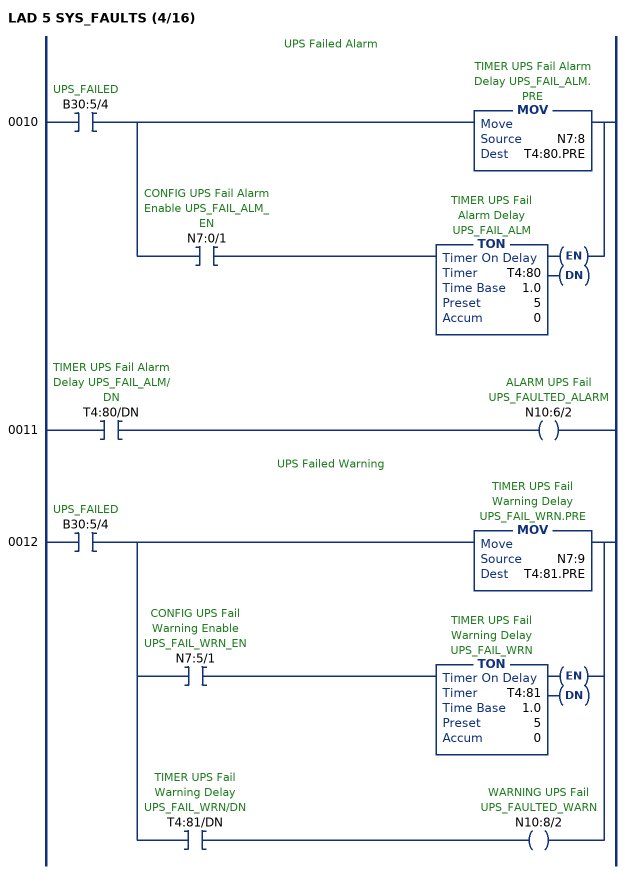
% Rung: 10 %
% UPS Failed Alarm %
SOR XIC B30:5/4 BST MOV N7:8 T4:80.PRE NXB XIC N7:0/1 TON T4:80 1.0 5 0 BND EOR
%   B30:5/4  UPS_FAILED %
%   N7:8  UPS_FAIL_ALM_DLY  "CONFIG UPS Fail Alarm Delay" %
%   T4:80  UPS_FAIL_ALM  "TIMER UPS Fail Alarm Delay" %
%   N7:0/1  UPS_FAIL_ALM_EN  "CONFIG UPS Fail Alarm Enable" %
% Rung: 11 %
SOR XIC T4:80/DN OTE N10:6/2 EOR
%   T4:80  UPS_FAIL_ALM  "TIMER UPS Fail Alarm Delay" %
%   N10:6/2  UPS_FAULTED_ALARM  "ALARM UPS Fail" %
% Rung: 12 %
% UPS Failed Warning %
SOR XIC B30:5/4 BST MOV N7:9 T4:81.PRE NXB XIC N7:5/1 TON T4:81 1.0 5 0 NXB XIC T4:81/DN OTE N10:8/2 BND EOR
%   B30:5/4  UPS_FAILED %
%   N7:9  UPS_FAIL_WRN_DLY  "CONFIG UPS Fail Warning Delay" %
%   T4:81  UPS_FAIL_WRN  "TIMER UPS Fail Warning Delay" %
%   N7:5/1  UPS_FAIL_WRN_EN  "CONFIG UPS Fail Warning Enable" %
%   N10:8/2  UPS_FAULTED_WARN  "WARNING UPS Fail" %

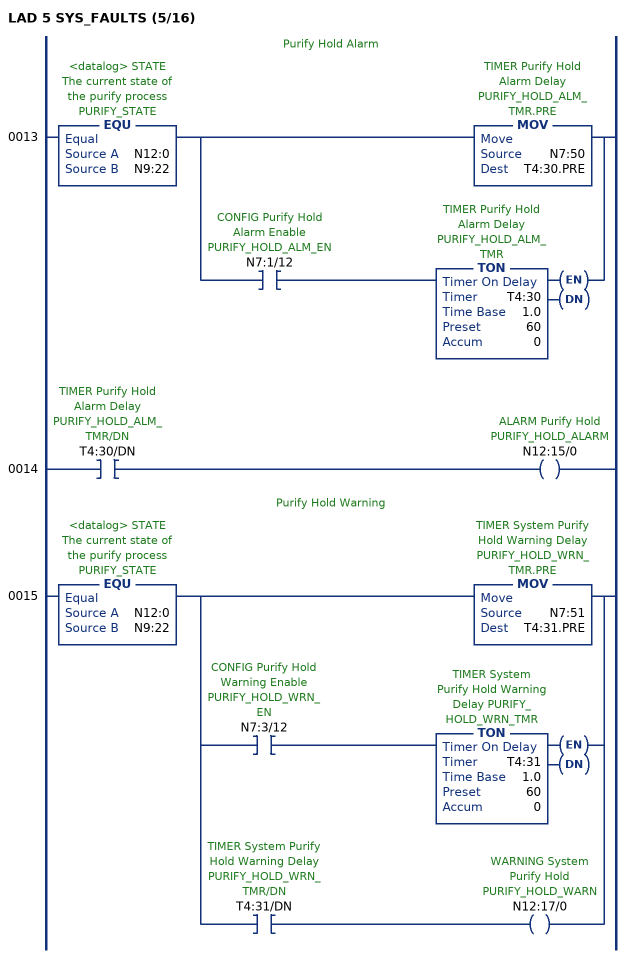
% Rung: 13 %
% Purify Hold Alarm %
SOR EQU N12:0 N9:22 BST MOV N7:50 T4:30.PRE NXB XIC N7:1/12 TON T4:30 1.0 60 0 BND EOR
%   N12:0  PURIFY_STATE  "<datalog> STATE The current state of the purify process" %
%   N9:22  PURIFY_HOLD  "STATE Purify Hold" %
%   N7:50  PURIFY_HOLD_ALM_DLY  "CONFIG Purify Hold Alarm Delay" %
%   T4:30  PURIFY_HOLD_ALM_TMR  "TIMER Purify Hold Alarm Delay" %
%   N7:1/12  PURIFY_HOLD_ALM_EN  "CONFIG Purify Hold Alarm Enable" %
% Rung: 14 %
SOR XIC T4:30/DN OTE N12:15/0 EOR
%   T4:30  PURIFY_HOLD_ALM_TMR  "TIMER Purify Hold Alarm Delay" %
%   N12:15/0  PURIFY_HOLD_ALARM  "ALARM Purify Hold" %
% Rung: 15 %
% Purify Hold Warning %
SOR EQU N12:0 N9:22 BST MOV N7:51 T4:31.PRE NXB XIC N7:3/12 TON T4:31 1.0 60 0 NXB XIC T4:31/DN OTE N12:17/0 BND EOR
%   N12:0  PURIFY_STATE  "<datalog> STATE The current state of the purify process" %
%   N9:22  PURIFY_HOLD  "STATE Purify Hold" %
%   N7:51  PURIFY_HOLD_WRN_DLY  "CONFIG Purify Hold Warning Delay" %
%   T4:31  PURIFY_HOLD_WRN_TMR  "TIMER System Purify Hold Warning Delay" %
%   N7:3/12  PURIFY_HOLD_WRN_EN  "CONFIG Purify Hold Warning Enable" %
%   N12:17/0  PURIFY_HOLD_WARN  "WARNING System Purify Hold" %

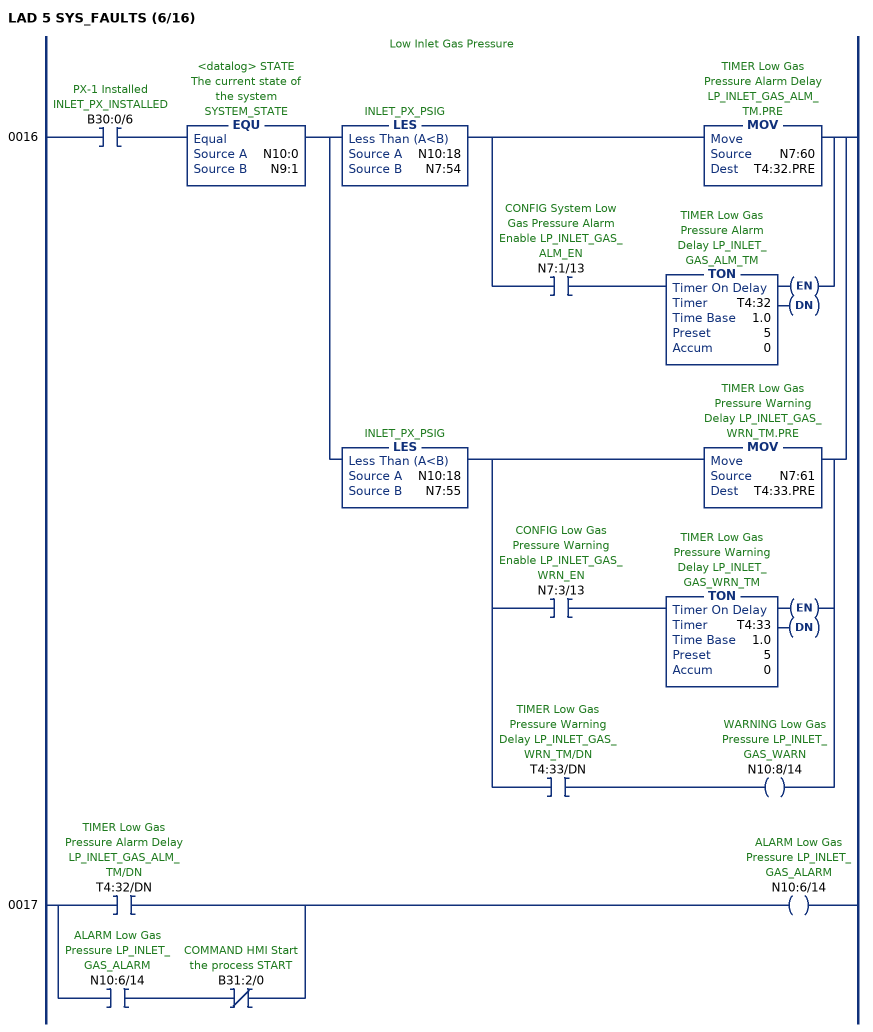
% Rung: 16 %
% Low Inlet Gas Pressure %
SOR XIC B30:0/6 EQU N10:0 N9:1 BST LES N10:18 N7:54 BST MOV N7:60 T4:32.PRE NXB XIC N7:1/13 TON T4:32 1.0 5 0 BND NXB LES N10:18 N7:55 BST MOV N7:61 T4:33.PRE NXB XIC N7:3/13 TON T4:33 1.0 5 0 NXB XIC T4:33/DN OTE N10:8/14 BND BND EOR
%   B30:0/6  INLET_PX_INSTALLED  "PX-1 Installed" %
%   N10:0  SYSTEM_STATE  "<datalog> STATE The current state of the system" %
%   N9:1  SYSTEM_PROCESS  "STATE System Process" %
%   N10:18  INLET_PX_PSIG %
%   N7:54  LP_INLET_GAS_ALM_SP  "CONFIG Gas Pressure Low Alarm Setpoint" %
%   N7:60  LP_INLET_GAS_ALM_DLY  "CONFIG Gas Pressure Low Alarm Delay" %
%   T4:32  LP_INLET_GAS_ALM_TM  "TIMER Low Gas Pressure Alarm Delay" %
%   N7:1/13  LP_INLET_GAS_ALM_EN  "CONFIG System Low Gas Pressure Alarm Enable" %
%   N7:55  LP_INLET_GAS_WRN_SP  "CONFIG Gas Pressure Low Warning Setpoint" %
%   N7:61  LP_INLET_GAS_WRN_DLY  "CONFIG Gas Pressure Low Warning Delay" %
%   T4:33  LP_INLET_GAS_WRN_TM  "TIMER Low Gas Pressure Warning Delay" %
%   N7:3/13  LP_INLET_GAS_WRN_EN  "CONFIG Low Gas Pressure Warning Enable" %
%   N10:8/14  LP_INLET_GAS_WARN  "WARNING Low Gas Pressure" %
% Rung: 17 %
SOR BST XIC T4:32/DN NXB XIC N10:6/14 XIO B31:2/0 BND OTE N10:6/14 EOR
%   T4:32  LP_INLET_GAS_ALM_TM  "TIMER Low Gas Pressure Alarm Delay" %
%   N10:6/14  LP_INLET_GAS_ALARM  "ALARM Low Gas Pressure" %
%   B31:2/0  START  "COMMAND HMI Start the process" %

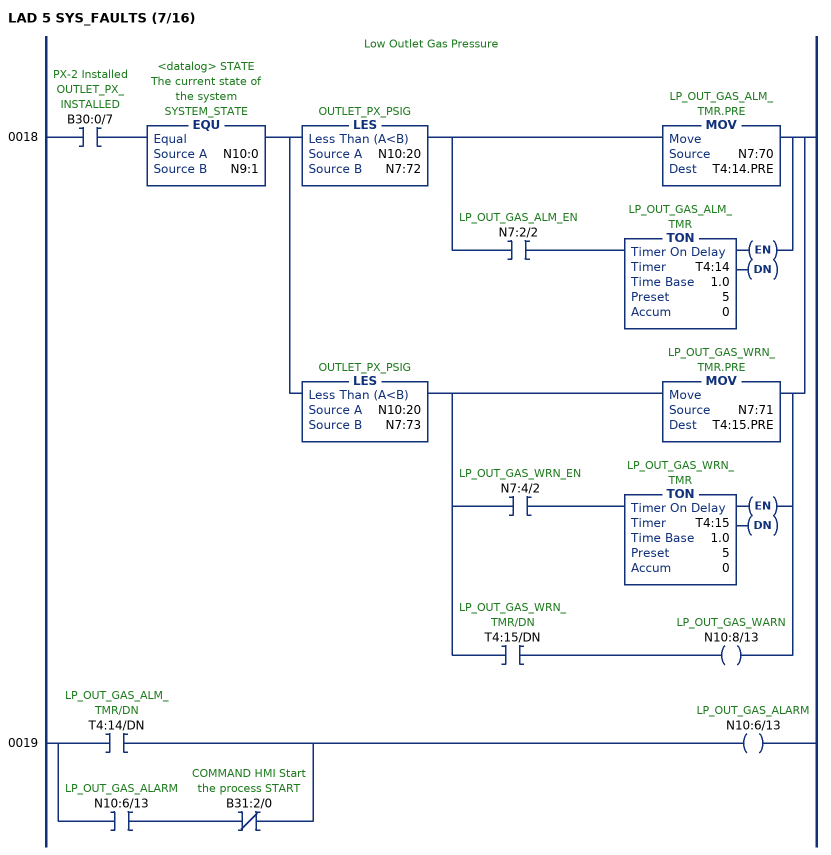
% Rung: 18 %
% Low Outlet Gas Pressure %
SOR XIC B30:0/7 EQU N10:0 N9:1 BST LES N10:20 N7:72 BST MOV N7:70 T4:14.PRE NXB XIC N7:2/2 TON T4:14 1.0 5 0 BND NXB LES N10:20 N7:73 BST MOV N7:71 T4:15.PRE NXB XIC N7:4/2 TON T4:15 1.0 5 0 NXB XIC T4:15/DN OTE N10:8/13 BND BND EOR
%   B30:0/7  OUTLET_PX_INSTALLED  "PX-2 Installed" %
%   N10:0  SYSTEM_STATE  "<datalog> STATE The current state of the system" %
%   N9:1  SYSTEM_PROCESS  "STATE System Process" %
%   N10:20  OUTLET_PX_PSIG %
%   N7:72  LP_OUT_GAS_ALM_SP %
%   N7:70  LP_OUT_GAS_ALM_DLY %
%   T4:14  LP_OUT_GAS_ALM_TMR %
%   N7:2/2  LP_OUT_GAS_ALM_EN %
%   N7:73  LP_OUT_GAS_WRN_SP %
%   N7:71  LP_OUT_GAS_WRN_DLY %
%   T4:15  LP_OUT_GAS_WRN_TMR %
%   N7:4/2  LP_OUT_GAS_WRN_EN %
%   N10:8/13  LP_OUT_GAS_WARN %
% Rung: 19 %
SOR BST XIC T4:14/DN NXB XIC N10:6/13 XIO B31:2/0 BND OTE N10:6/13 EOR
%   T4:14  LP_OUT_GAS_ALM_TMR %
%   N10:6/13  LP_OUT_GAS_ALARM %
%   B31:2/0  START  "COMMAND HMI Start the process" %

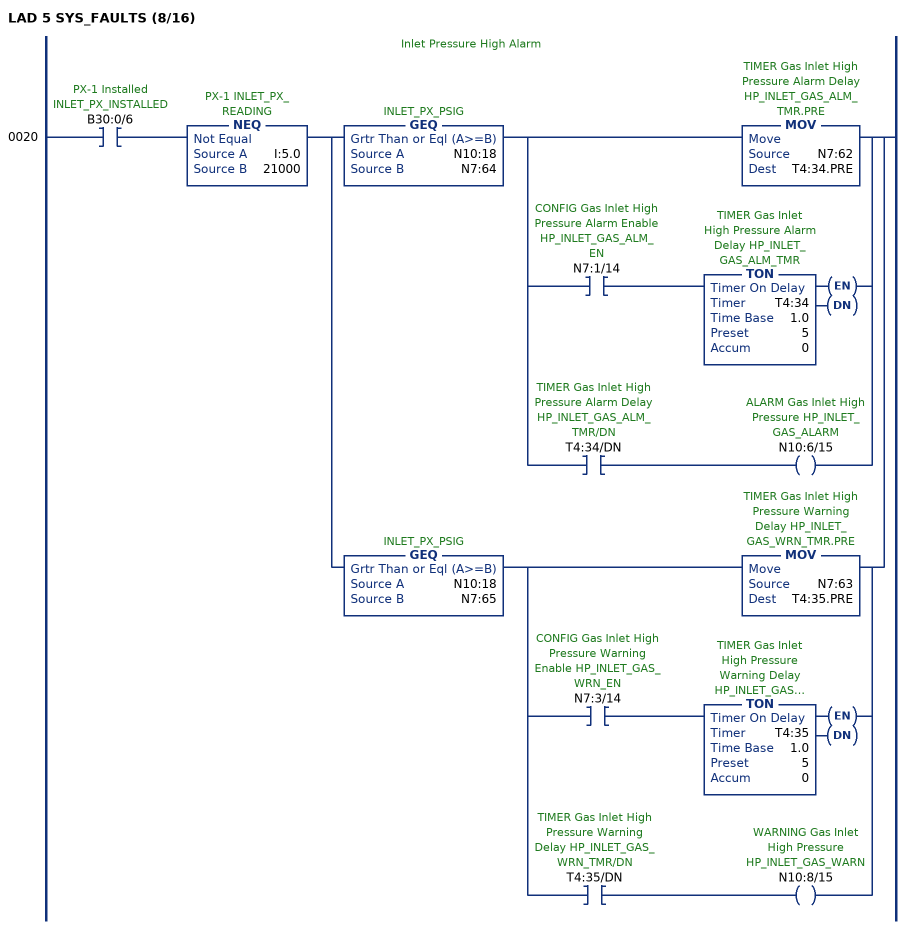
% Rung: 20 %
% Inlet Pressure High Alarm %
SOR XIC B30:0/6 NEQ I:5.0 21000 BST GEQ N10:18 N7:64 BST MOV N7:62 T4:34.PRE NXB XIC N7:1/14 TON T4:34 1.0 5 0 NXB XIC T4:34/DN OTE N10:6/15 BND NXB GEQ N10:18 N7:65 BST MOV N7:63 T4:35.PRE NXB XIC N7:3/14 TON T4:35 1.0 5 0 NXB XIC T4:35/DN OTE N10:8/15 BND BND EOR
%   B30:0/6  INLET_PX_INSTALLED  "PX-1 Installed" %
%   I:5.0  INLET_PX_READING  "PX-1" %
%   N10:18  INLET_PX_PSIG %
%   N7:64  HP_INLET_GAS_ALM_SP  "CONFIG Gas Inlet High Pressure Alarm Setpoint" %
%   N7:62  HP_INLET_GAS_ALM_DLY  "CONFIG Gas Inlet High Pressure Alarm Delay" %
%   T4:34  HP_INLET_GAS_ALM_TMR  "TIMER Gas Inlet High Pressure Alarm Delay" %
%   N7:1/14  HP_INLET_GAS_ALM_EN  "CONFIG Gas Inlet High Pressure Alarm Enable" %
%   N10:6/15  HP_INLET_GAS_ALARM  "ALARM Gas Inlet High Pressure" %
%   N7:65  HP_INLET_GAS_WRN_SP  "CONFIG Gas Inlet High Pressure Warning Setpoint" %
%   N7:63  HP_INLET_GAS_WRN_DLY  "CONFIG Gas Inlet High Pressure Warning Delay" %
%   T4:35  HP_INLET_GAS_WRN_TMR  "TIMER Gas Inlet High Pressure Warning Delay" %
%   N7:3/14  HP_INLET_GAS_WRN_EN  "CONFIG Gas Inlet High Pressure Warning Enable" %
%   N10:8/15  HP_INLET_GAS_WARN  "WARNING Gas Inlet High Pressure" %

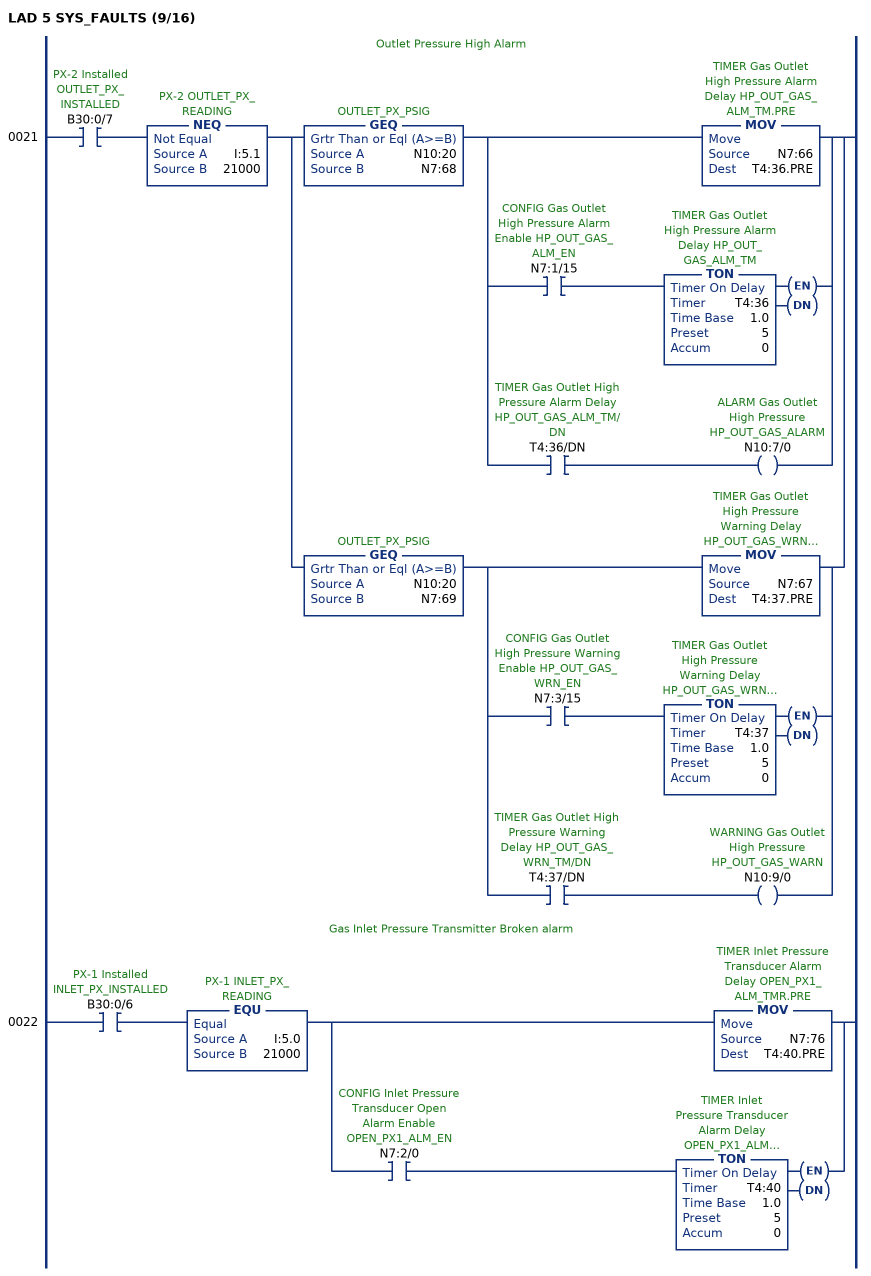
% Rung: 21 %
% Outlet Pressure High Alarm %
SOR XIC B30:0/7 NEQ I:5.1 21000 BST GEQ N10:20 N7:68 BST MOV N7:66 T4:36.PRE NXB XIC N7:1/15 TON T4:36 1.0 5 0 NXB XIC T4:36/DN OTE N10:7/0 BND NXB GEQ N10:20 N7:69 BST MOV N7:67 T4:37.PRE NXB XIC N7:3/15 TON T4:37 1.0 5 0 NXB XIC T4:37/DN OTE N10:9/0 BND BND EOR
%   B30:0/7  OUTLET_PX_INSTALLED  "PX-2 Installed" %
%   I:5.1  OUTLET_PX_READING  "PX-2" %
%   N10:20  OUTLET_PX_PSIG %
%   N7:68  HP_OUT_GAS_ALM_SP  "CONFIG Gas Outlet High Pressure Alarm Setpoint" %
%   N7:66  HP_OUT_GAS_ALM_DLY  "CONFIG Gas Outlet High Pressure Alarm Deley" %
%   T4:36  HP_OUT_GAS_ALM_TM  "TIMER Gas Outlet High Pressure Alarm Delay" %
%   N7:1/15  HP_OUT_GAS_ALM_EN  "CONFIG Gas Outlet High Pressure Alarm Enable" %
%   N10:7/0  HP_OUT_GAS_ALARM  "ALARM Gas Outlet High Pressure" %
%   N7:69  HP_OUT_GAS_WRN_SP  "CONFIG Gas Outlet High Pressure Warning Setpoint" %
%   N7:67  HP_OUT_GAS_WRN_DLY  "CONFIG Gas Outlet High Pressure Warning Delay" %
%   T4:37  HP_OUT_GAS_WRN_TM  "TIMER Gas Outlet High Pressure Warning Delay" %
%   N7:3/15  HP_OUT_GAS_WRN_EN  "CONFIG Gas Outlet High Pressure Warning Enable" %
%   N10:9/0  HP_OUT_GAS_WARN  "WARNING Gas Outlet High Pressure" %
% Rung: 22 %
% Gas Inlet Pressure Transmitter Broken alarm %
SOR XIC B30:0/6 EQU I:5.0 21000 BST MOV N7:76 T4:40.PRE NXB XIC N7:2/0 TON T4:40 1.0 5 0 BND EOR
%   B30:0/6  INLET_PX_INSTALLED  "PX-1 Installed" %
%   I:5.0  INLET_PX_READING  "PX-1" %
%   N7:76  OPEN_PX1_ALM_DLY  "CONFIG Inlet Pressure Transducer Open Alarm Delay" %
%   T4:40  OPEN_PX1_ALM_TMR  "TIMER Inlet Pressure Transducer Alarm Delay" %
%   N7:2/0  OPEN_PX1_ALM_EN  "CONFIG Inlet Pressure Transducer Open Alarm Enable" %

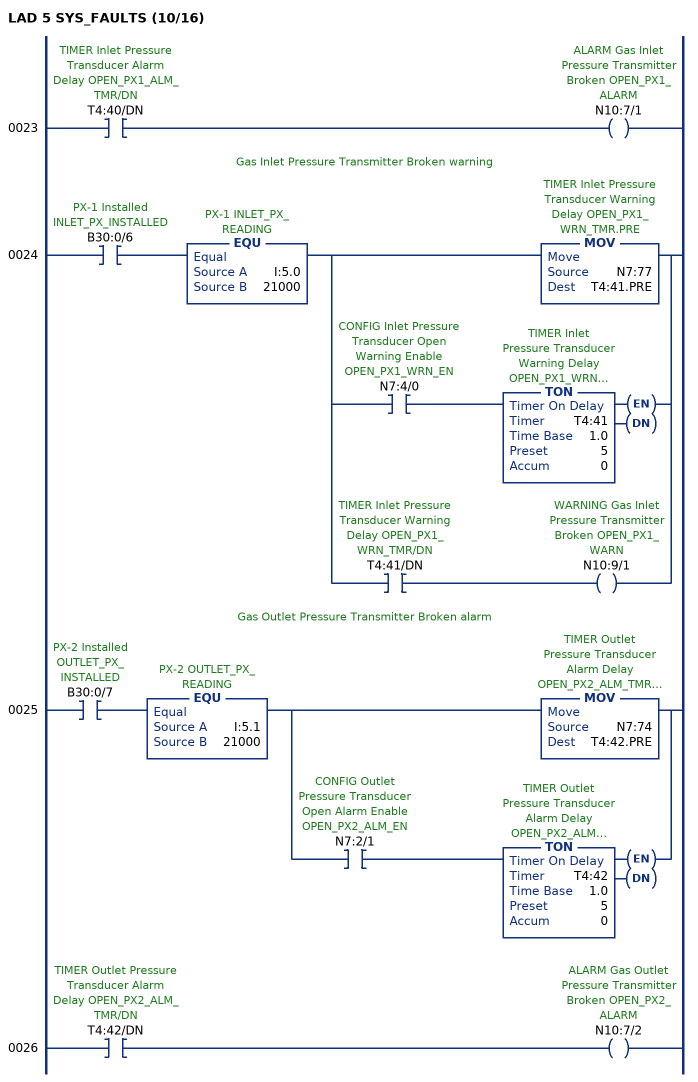
% Rung: 23 %
SOR XIC T4:40/DN OTE N10:7/1 EOR
%   T4:40  OPEN_PX1_ALM_TMR  "TIMER Inlet Pressure Transducer Alarm Delay" %
%   N10:7/1  OPEN_PX1_ALARM  "ALARM Gas Inlet Pressure Transmitter Broken" %
% Rung: 24 %
% Gas Inlet Pressure Transmitter Broken warning %
SOR XIC B30:0/6 EQU I:5.0 21000 BST MOV N7:77 T4:41.PRE NXB XIC N7:4/0 TON T4:41 1.0 5 0 NXB XIC T4:41/DN OTE N10:9/1 BND EOR
%   B30:0/6  INLET_PX_INSTALLED  "PX-1 Installed" %
%   I:5.0  INLET_PX_READING  "PX-1" %
%   N7:77  OPEN_PX1_WRN_DLY  "CONFIG Inlet Pressure Transducer Open Warning Delay" %
%   T4:41  OPEN_PX1_WRN_TMR  "TIMER Inlet Pressure Transducer Warning Delay" %
%   N7:4/0  OPEN_PX1_WRN_EN  "CONFIG Inlet Pressure Transducer Open Warning Enable" %
%   N10:9/1  OPEN_PX1_WARN  "WARNING Gas Inlet Pressure Transmitter Broken" %
% Rung: 25 %
% Gas Outlet Pressure Transmitter Broken alarm %
SOR XIC B30:0/7 EQU I:5.1 21000 BST MOV N7:74 T4:42.PRE NXB XIC N7:2/1 TON T4:42 1.0 5 0 BND EOR
%   B30:0/7  OUTLET_PX_INSTALLED  "PX-2 Installed" %
%   I:5.1  OUTLET_PX_READING  "PX-2" %
%   N7:74  OPEN_PX2_ALM_DLY  "CONFIG Outlet Pressure Transducer Open Alarm Delay" %
%   T4:42  OPEN_PX2_ALM_TMR  "TIMER Outlet Pressure Transducer Alarm Delay" %
%   N7:2/1  OPEN_PX2_ALM_EN  "CONFIG Outlet Pressure Transducer Open Alarm Enable" %
% Rung: 26 %
SOR XIC T4:42/DN OTE N10:7/2 EOR
%   T4:42  OPEN_PX2_ALM_TMR  "TIMER Outlet Pressure Transducer Alarm Delay" %
%   N10:7/2  OPEN_PX2_ALARM  "ALARM Gas Outlet Pressure Transmitter Broken" %

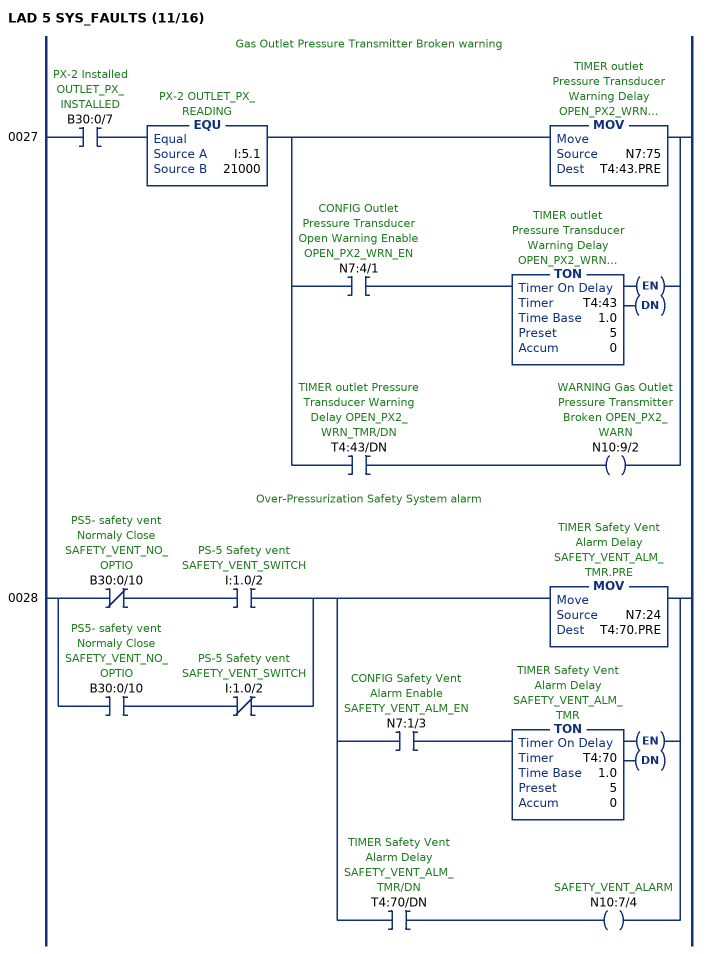
% Rung: 27 %
% Gas Outlet Pressure Transmitter Broken warning %
SOR XIC B30:0/7 EQU I:5.1 21000 BST MOV N7:75 T4:43.PRE NXB XIC N7:4/1 TON T4:43 1.0 5 0 NXB XIC T4:43/DN OTE N10:9/2 BND EOR
%   B30:0/7  OUTLET_PX_INSTALLED  "PX-2 Installed" %
%   I:5.1  OUTLET_PX_READING  "PX-2" %
%   N7:75  OPEN_PX2_WRN_DLY  "CONFIG Outlet Pressure Transducer Open Warning Delay" %
%   T4:43  OPEN_PX2_WRN_TMR  "TIMER outlet Pressure Transducer Warning Delay" %
%   N7:4/1  OPEN_PX2_WRN_EN  "CONFIG Outlet Pressure Transducer Open Warning Enable" %
%   N10:9/2  OPEN_PX2_WARN  "WARNING Gas Outlet Pressure Transmitter Broken" %
% Rung: 28 %
% Over-Pressurization Safety System alarm %
SOR BST XIO B30:0/10 XIC I:1.0/2 NXB XIC B30:0/10 XIO I:1.0/2 BND BST MOV N7:24 T4:70.PRE NXB XIC N7:1/3 TON T4:70 1.0 5 0 NXB XIC T4:70/DN OTE N10:7/4 BND EOR
%   B30:0/10  SAFETY_VENT_NO_OPTIO  "PS5- safety vent Normaly Close" %
%   I:1.0/2  SAFETY_VENT_SWITCH  "PS-5 Safety vent" %
%   N7:24  SAFETY_VENT_ALM_DLY  "CONFIG Safety Vent Alarm Delay" %
%   T4:70  SAFETY_VENT_ALM_TMR  "TIMER Safety Vent Alarm Delay" %
%   N7:1/3  SAFETY_VENT_ALM_EN  "CONFIG Safety Vent Alarm Enable" %
%   N10:7/4  SAFETY_VENT_ALARM %

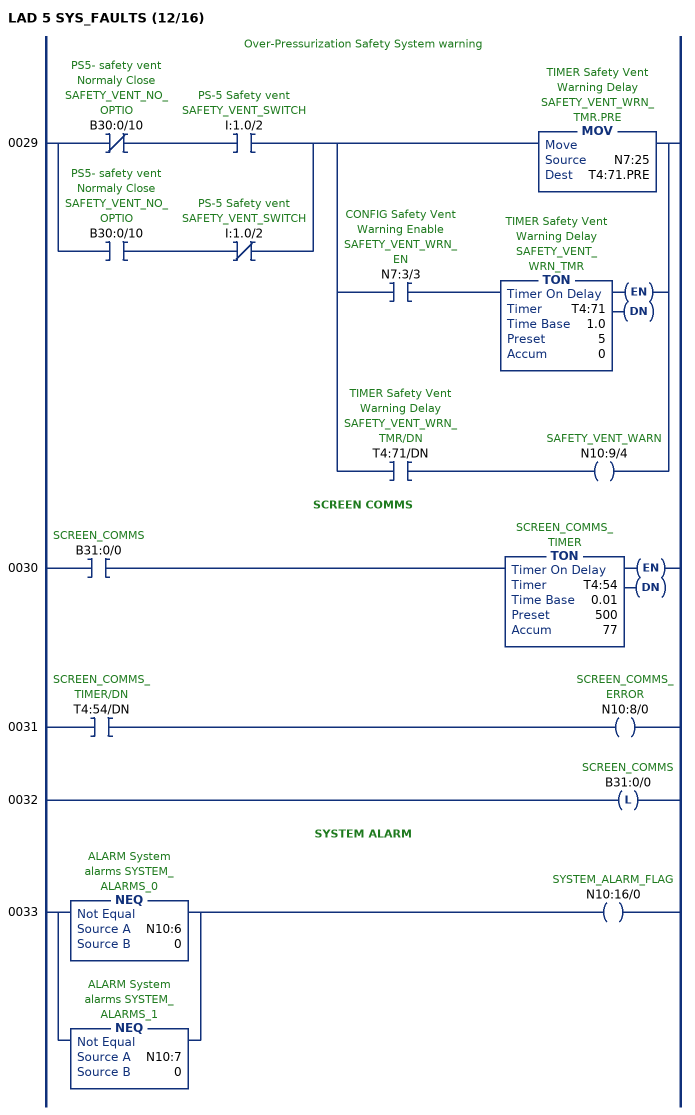
% Rung: 29 %
% Over-Pressurization Safety System warning %
SOR BST XIO B30:0/10 XIC I:1.0/2 NXB XIC B30:0/10 XIO I:1.0/2 BND BST MOV N7:25 T4:71.PRE NXB XIC N7:3/3 TON T4:71 1.0 5 0 NXB XIC T4:71/DN OTE N10:9/4 BND EOR
%   B30:0/10  SAFETY_VENT_NO_OPTIO  "PS5- safety vent Normaly Close" %
%   I:1.0/2  SAFETY_VENT_SWITCH  "PS-5 Safety vent" %
%   N7:25  SAFETY_VENT_WRN_DLY  "CONFIG Safety Vent Warning Delay" %
%   T4:71  SAFETY_VENT_WRN_TMR  "TIMER Safety Vent Warning Delay" %
%   N7:3/3  SAFETY_VENT_WRN_EN  "CONFIG Safety Vent Warning Enable" %
%   N10:9/4  SAFETY_VENT_WARN %
% Rung: 30 %
% TITLE: SCREEN COMMS %
SOR XIC B31:0/0 TON T4:54 0.01 500 77 EOR
%   B31:0/0  SCREEN_COMMS %
%   T4:54  SCREEN_COMMS_TIMER %
% Rung: 31 %
SOR XIC T4:54/DN OTE N10:8/0 EOR
%   T4:54  SCREEN_COMMS_TIMER %
%   N10:8/0  SCREEN_COMMS_ERROR %
% Rung: 32 %
SOR OTL B31:0/0 EOR
%   B31:0/0  SCREEN_COMMS %
% Rung: 33 %
% TITLE: SYSTEM ALARM %
SOR BST NEQ N10:6 0 NXB NEQ N10:7 0 BND OTE N10:16/0 EOR
%   N10:6  SYSTEM_ALARMS_0  "ALARM System alarms" %
%   N10:7  SYSTEM_ALARMS_1  "ALARM System alarms" %
%   N10:16/0  SYSTEM_ALARM_FLAG %

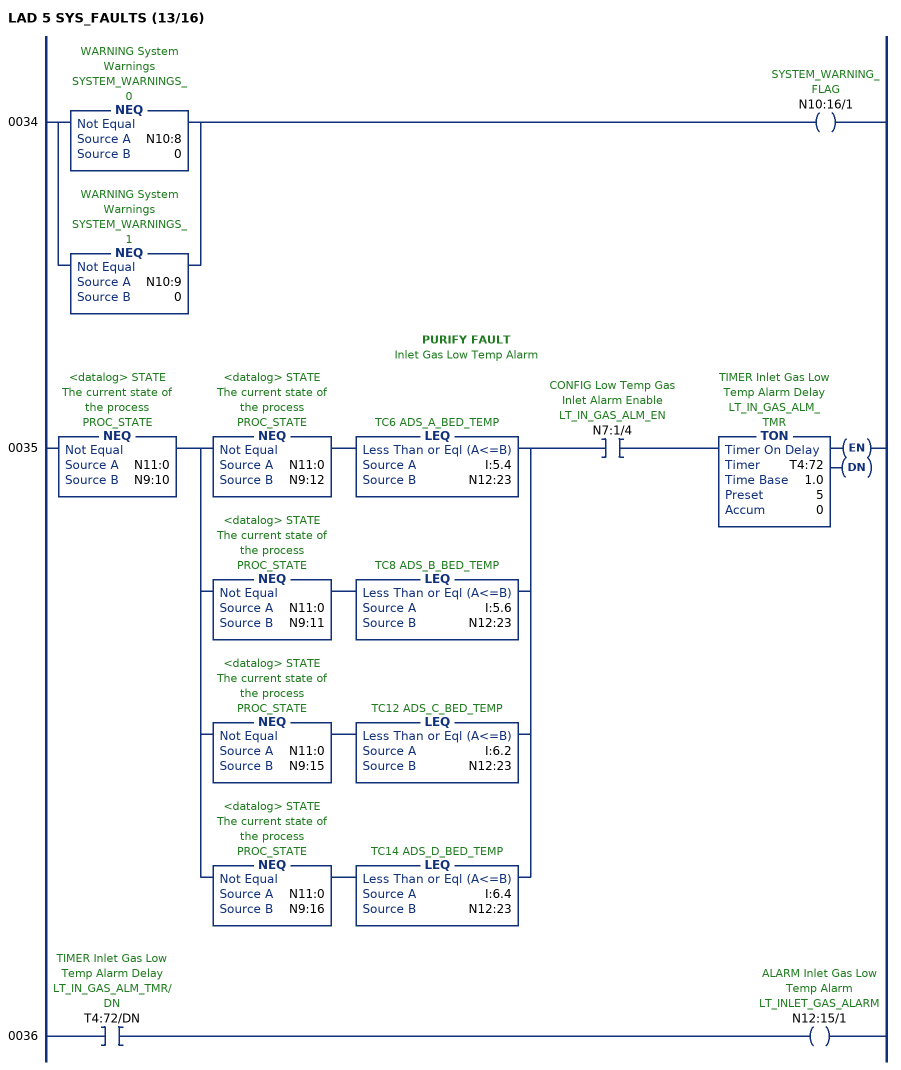
% Rung: 34 %
SOR BST NEQ N10:8 0 NXB NEQ N10:9 0 BND OTE N10:16/1 EOR
%   N10:8  SYSTEM_WARNINGS_0  "WARNING System Warnings" %
%   N10:9  SYSTEM_WARNINGS_1  "WARNING System Warnings" %
%   N10:16/1  SYSTEM_WARNING_FLAG %
% Rung: 35 %
% TITLE: PURIFY FAULT %
% Inlet Gas Low Temp Alarm %
SOR NEQ N11:0 N9:10 BST NEQ N11:0 N9:12 LEQ I:5.4 N12:23 NXB NEQ N11:0 N9:11 LEQ I:5.6 N12:23 NXB NEQ N11:0 N9:15 LEQ I:6.2 N12:23 NXB NEQ N11:0 N9:16 LEQ I:6.4 N12:23 BND XIC N7:1/4 TON T4:72 1.0 5 0 EOR
%   N11:0  PROC_STATE  "<datalog> STATE The current state of the process" %
%   N9:10  PROCESS_STANDBY  "STATE Process Standby" %
%   N9:12  PROC_REGEN_A  "STATE Process Regen A" %
%   I:5.4  ADS_A_BED_TEMP  "TC6" %
%   N12:23  LT_INLET_GAS_ALM_SP  "CONFIG Low Temp Inlet Gas Alarm Setpoint" %
%   N9:11  PROC_REGEN_B  "STATE Process Regen B" %
%   I:5.6  ADS_B_BED_TEMP  "TC8" %
%   N9:15  PROC_REGEN_C  "STATE Process Regen C" %
%   I:6.2  ADS_C_BED_TEMP  "TC12" %
%   N9:16  PROC_REGEN_D  "STATE Process Regen D" %
%   I:6.4  ADS_D_BED_TEMP  "TC14" %
%   N7:1/4  LT_IN_GAS_ALM_EN  "CONFIG Low Temp Gas Inlet Alarm Enable" %
%   T4:72  LT_IN_GAS_ALM_TMR  "TIMER Inlet Gas Low Temp Alarm Delay" %
% Rung: 36 %
SOR XIC T4:72/DN OTE N12:15/1 EOR
%   T4:72  LT_IN_GAS_ALM_TMR  "TIMER Inlet Gas Low Temp Alarm Delay" %
%   N12:15/1  LT_INLET_GAS_ALARM  "ALARM Inlet Gas Low Temp Alarm" %

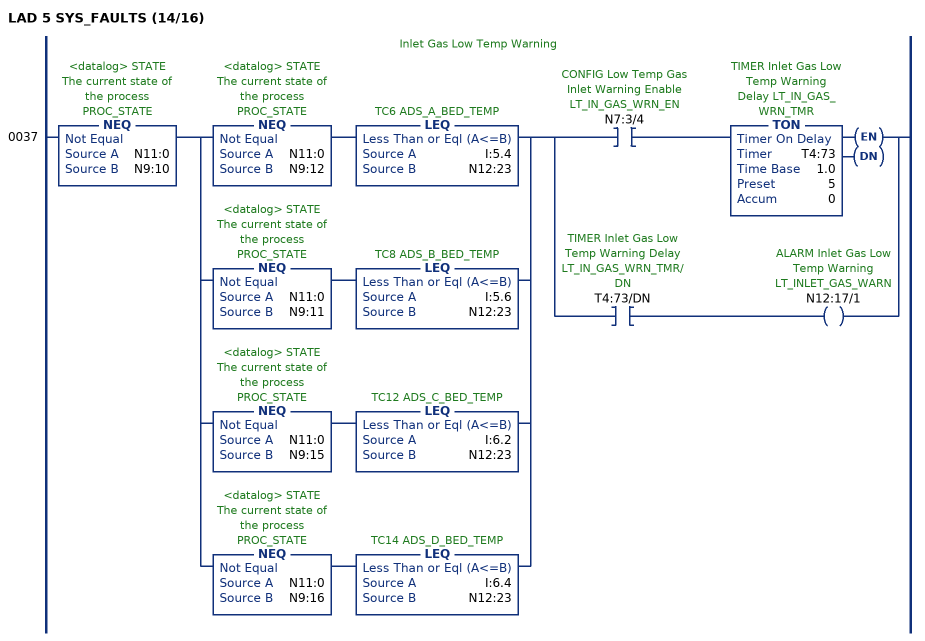
% Rung: 37 %
% Inlet Gas Low Temp Warning %
SOR NEQ N11:0 N9:10 BST NEQ N11:0 N9:12 LEQ I:5.4 N12:23 NXB NEQ N11:0 N9:11 LEQ I:5.6 N12:23 NXB NEQ N11:0 N9:15 LEQ I:6.2 N12:23 NXB NEQ N11:0 N9:16 LEQ I:6.4 N12:23 BND BST XIC N7:3/4 TON T4:73 1.0 5 0 NXB XIC T4:73/DN OTE N12:17/1 BND EOR
%   N11:0  PROC_STATE  "<datalog> STATE The current state of the process" %
%   N9:10  PROCESS_STANDBY  "STATE Process Standby" %
%   N9:12  PROC_REGEN_A  "STATE Process Regen A" %
%   I:5.4  ADS_A_BED_TEMP  "TC6" %
%   N12:23  LT_INLET_GAS_ALM_SP  "CONFIG Low Temp Inlet Gas Alarm Setpoint" %
%   N9:11  PROC_REGEN_B  "STATE Process Regen B" %
%   I:5.6  ADS_B_BED_TEMP  "TC8" %
%   N9:15  PROC_REGEN_C  "STATE Process Regen C" %
%   I:6.2  ADS_C_BED_TEMP  "TC12" %
%   N9:16  PROC_REGEN_D  "STATE Process Regen D" %
%   I:6.4  ADS_D_BED_TEMP  "TC14" %
%   N7:3/4  LT_IN_GAS_WRN_EN  "CONFIG Low Temp Gas Inlet Warning Enable" %
%   T4:73  LT_IN_GAS_WRN_TMR  "TIMER Inlet Gas Low Temp Warning Delay" %
%   N12:17/1  LT_INLET_GAS_WARN  "ALARM Inlet Gas Low Temp Warning" %

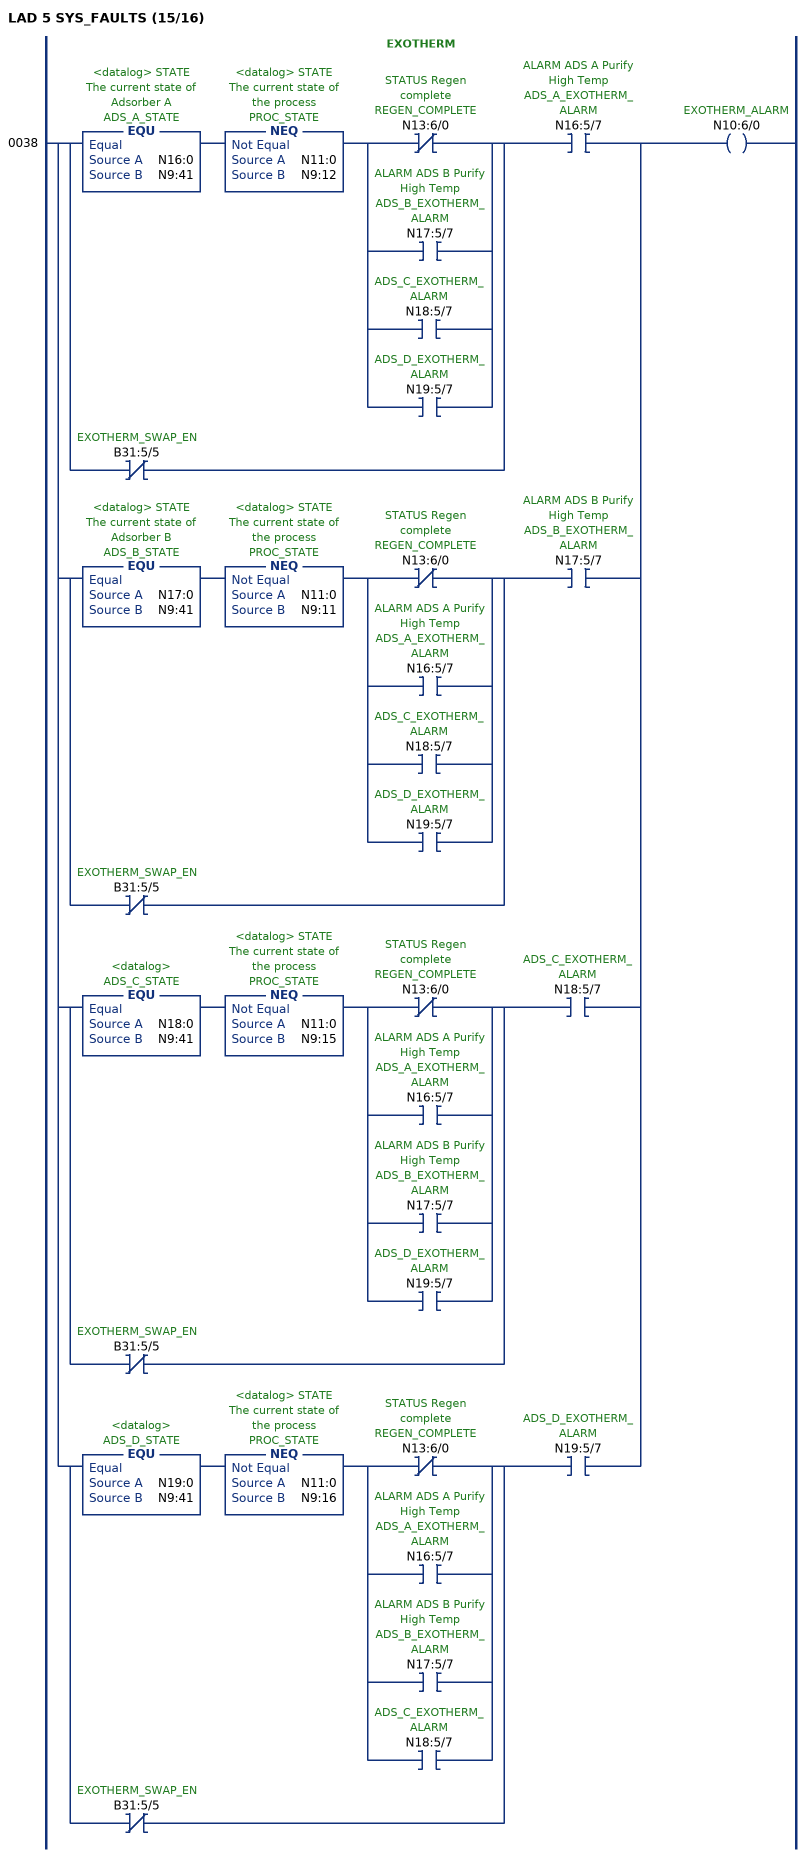
% Rung: 38 %
% TITLE: EXOTHERM %
SOR BST BST EQU N16:0 N9:41 NEQ N11:0 N9:12 BST XIO N13:6/0 NXB XIC N17:5/7 NXB XIC N18:5/7 NXB XIC N19:5/7 BND NXB XIO B31:5/5 BND XIC N16:5/7 NXB BST EQU N17:0 N9:41 NEQ N11:0 N9:11 BST XIO N13:6/0 NXB XIC N16:5/7 NXB XIC N18:5/7 NXB XIC N19:5/7 BND NXB XIO B31:5/5 BND XIC N17:5/7 NXB BST EQU N18:0 N9:41 NEQ N11:0 N9:15 BST XIO N13:6/0 NXB XIC N16:5/7 NXB XIC N17:5/7 NXB XIC N19:5/7 BND NXB XIO B31:5/5 BND XIC N18:5/7 NXB BST EQU N19:0 N9:41 NEQ N11:0 N9:16 BST XIO N13:6/0 NXB XIC N16:5/7 NXB XIC N17:5/7 NXB XIC N18:5/7 BND NXB XIO B31:5/5 BND XIC N19:5/7 BND OTE N10:6/0 EOR
%   N16:0  ADS_A_STATE  "<datalog> STATE The current state of Adsorber A" %
%   N9:41  ADS_PURIFY  "STATE ADS Purify" %
%   N11:0  PROC_STATE  "<datalog> STATE The current state of the process" %
%   N9:12  PROC_REGEN_A  "STATE Process Regen A" %
%   N13:6/0  REGEN_COMPLETE  "STATUS Regen complete" %
%   N17:5/7  ADS_B_EXOTHERM_ALARM  "ALARM ADS B Purify High Temp" %
%   N18:5/7  ADS_C_EXOTHERM_ALARM %
%   N19:5/7  ADS_D_EXOTHERM_ALARM %
%   B31:5/5  EXOTHERM_SWAP_EN %
%   N16:5/7  ADS_A_EXOTHERM_ALARM  "ALARM ADS A Purify High Temp" %
%   N17:0  ADS_B_STATE  "<datalog> STATE The current state of Adsorber B" %
%   N9:11  PROC_REGEN_B  "STATE Process Regen B" %
%   N18:0  ADS_C_STATE  "<datalog>" %
%   N9:15  PROC_REGEN_C  "STATE Process Regen C" %
%   N19:0  ADS_D_STATE  "<datalog>" %
%   N9:16  PROC_REGEN_D  "STATE Process Regen D" %
%   N10:6/0  EXOTHERM_ALARM %

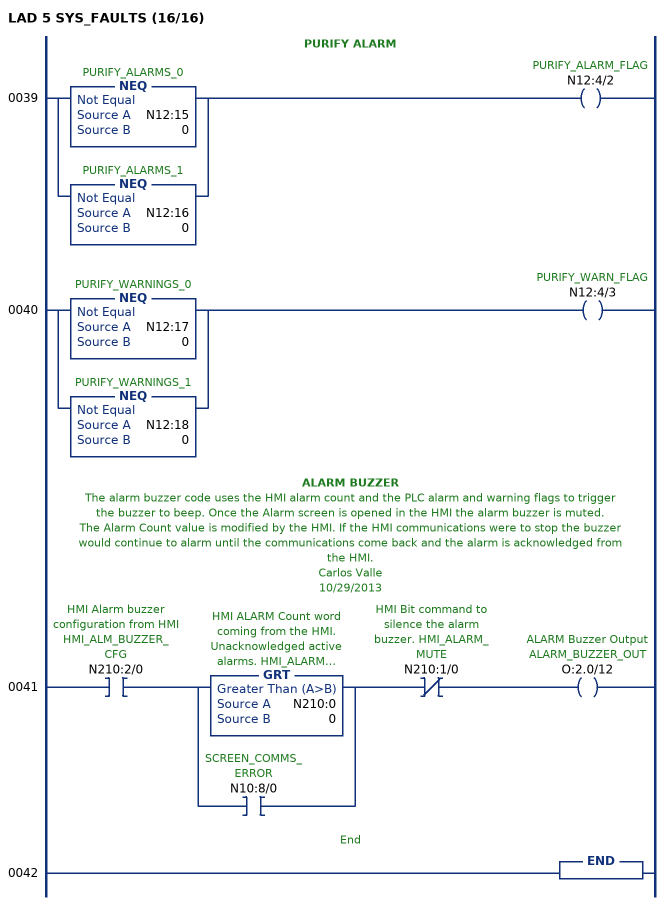
% Rung: 39 %
% TITLE: PURIFY ALARM %
SOR BST NEQ N12:15 0 NXB NEQ N12:16 0 BND OTE N12:4/2 EOR
%   N12:15  PURIFY_ALARMS_0 %
%   N12:16  PURIFY_ALARMS_1 %
%   N12:4/2  PURIFY_ALARM_FLAG %
% Rung: 40 %
SOR BST NEQ N12:17 0 NXB NEQ N12:18 0 BND OTE N12:4/3 EOR
%   N12:17  PURIFY_WARNINGS_0 %
%   N12:18  PURIFY_WARNINGS_1 %
%   N12:4/3  PURIFY_WARN_FLAG %
% Rung: 41 %
% TITLE: ALARM BUZZER %
% The alarm buzzer code uses the HMI alarm count and the PLC alarm and warning flags to trigger the buzzer to beep. Once the Alarm screen is opened in the HMI the alarm buzzer is muted.
% The Alarm Count value is modified by the HMI. If the HMI communications were to stop the buzzer would continue to alarm until the communications come back and the alarm is acknowledged from the HMI.
% Carlos Valle
% 10/29/2013 %
SOR XIC N210:2/0 BST GRT N210:0 0 NXB XIC N10:8/0 BND XIO N210:1/0 OTE O:2.0/12 EOR
%   N210:2/0  HMI_ALM_BUZZER_CFG  "HMI Alarm buzzer configuration from HMI" %
%   N210:0  HMI_ALARM_COUNT  "HMI ALARM Count word coming from the HMI. Unacknowledged active alarms." %
%   N10:8/0  SCREEN_COMMS_ERROR %
%   N210:1/0  HMI_ALARM_MUTE  "HMI Bit command to silence the alarm buzzer." %
%   O:2.0/12  ALARM_BUZZER_OUT  "ALARM Buzzer Output" %
% Rung: 42 %
% End %
SOR END EOR

LADDER 6 "SYSTEM"    % Controls the system %
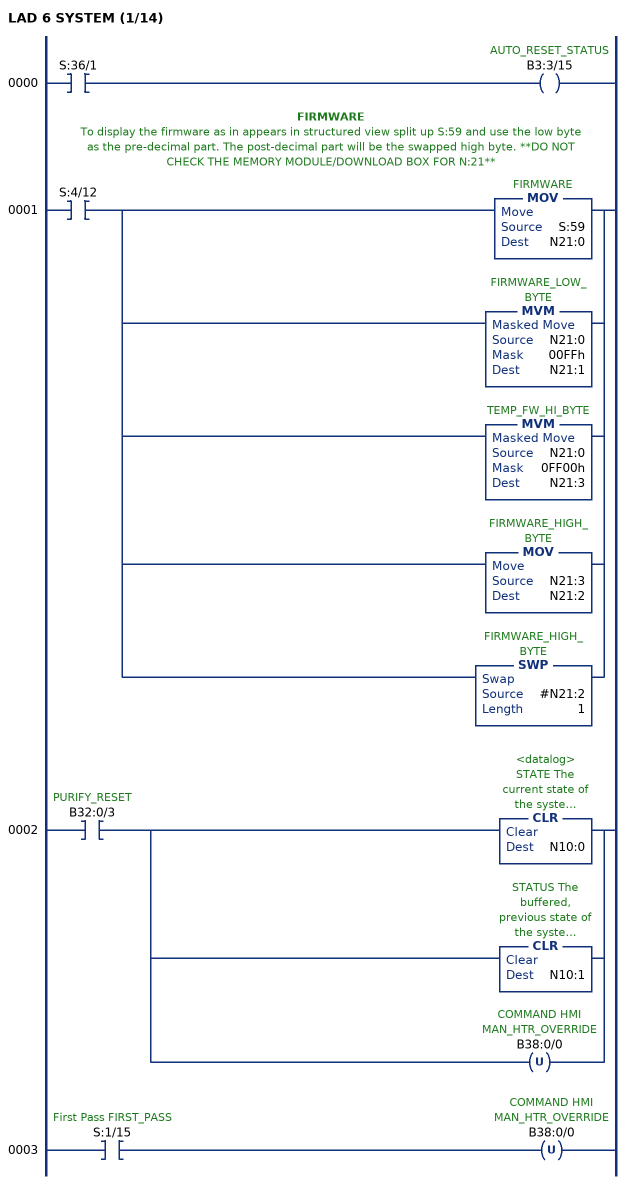
% Rung: 0 %
SOR XIC S:36/1 OTE B3:3/15 EOR
%   B3:3/15  AUTO_RESET_STATUS %
% Rung: 1 %
% TITLE: FIRMWARE %
% To display the firmware as in appears in structured view split up S:59 and use the low byte as the pre-decimal part. The post-decimal part will be the swapped high byte. **DO NOT CHECK THE MEMORY MODULE/DOWNLOAD BOX FOR N:21** %
SOR XIC S:4/12 BST MOV S:59 N21:0 NXB MVM N21:0 00FFh N21:1 NXB MVM N21:0 0FF00h N21:3 NXB MOV N21:3 N21:2 NXB SWP #N21:2 1 BND EOR
%   S:59  "Operating System FRN" %
%   N21:0  FIRMWARE %
%   N21:1  FIRMWARE_LOW_BYTE %
%   N21:3  TEMP_FW_HI_BYTE %
%   N21:2  FIRMWARE_HIGH_BYTE %
% Rung: 2 %
SOR XIC B32:0/3 BST CLR N10:0 NXB CLR N10:1 NXB OTU B38:0/0 BND EOR
%   B32:0/3  PURIFY_RESET %
%   N10:0  SYSTEM_STATE  "<datalog> STATE The current state of the system" %
%   N10:1  SYSTEM_BUFFER  "STATUS The buffered, previous state of the system" %
%   B38:0/0  MAN_HTR_OVERRIDE  "COMMAND HMI" %
% Rung: 3 %
SOR XIC S:1/15 OTU B38:0/0 EOR
%   S:1/15  FIRST_PASS  "First Pass" %
%   B38:0/0  MAN_HTR_OVERRIDE  "COMMAND HMI" %

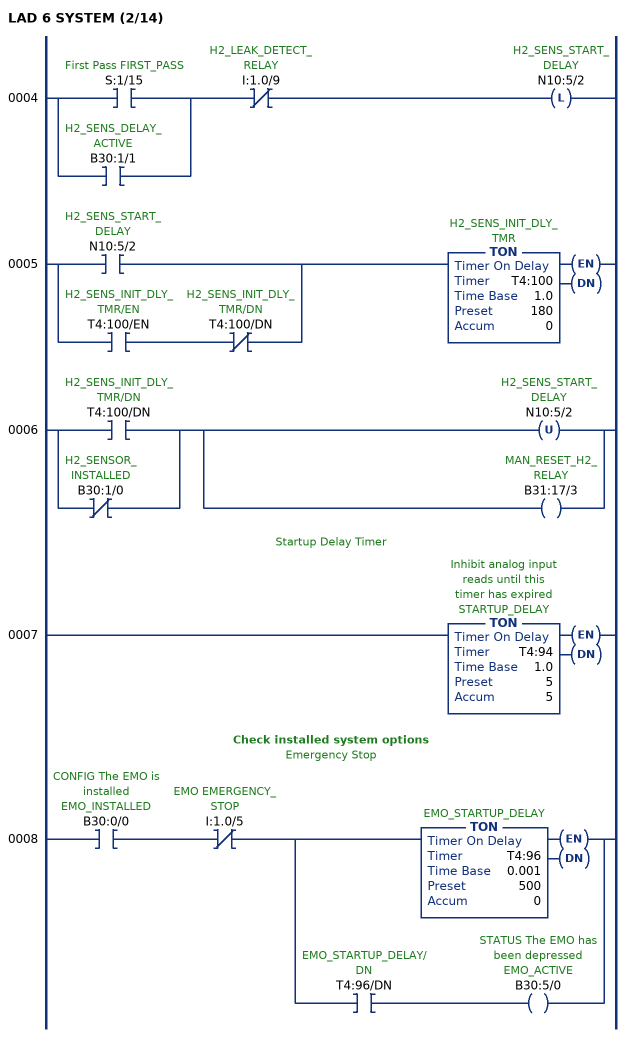
% Rung: 4 %
SOR BST XIC S:1/15 NXB XIC B30:1/1 BND XIO I:1.0/9 OTL N10:5/2 EOR
%   S:1/15  FIRST_PASS  "First Pass" %
%   B30:1/1  H2_SENS_DELAY_ACTIVE %
%   I:1.0/9  H2_LEAK_DETECT_RELAY %
%   N10:5/2  H2_SENS_START_DELAY %
% Rung: 5 %
SOR BST XIC N10:5/2 NXB XIC T4:100/EN XIO T4:100/DN BND TON T4:100 1.0 180 0 EOR
%   N10:5/2  H2_SENS_START_DELAY %
%   T4:100  H2_SENS_INIT_DLY_TMR %
% Rung: 6 %
SOR BST XIC T4:100/DN NXB XIO B30:1/0 BND BST OTU N10:5/2 NXB OTE B31:17/3 BND EOR
%   T4:100  H2_SENS_INIT_DLY_TMR %
%   B30:1/0  H2_SENSOR_INSTALLED %
%   N10:5/2  H2_SENS_START_DELAY %
%   B31:17/3  MAN_RESET_H2_RELAY %
% Rung: 7 %
% Startup Delay Timer %
SOR TON T4:94 1.0 5 5 EOR
%   T4:94  STARTUP_DELAY  "Inhibit analog input reads until this timer has expired" %
% Rung: 8 %
% TITLE: Check installed system options %
% Emergency Stop %
SOR XIC B30:0/0 XIO I:1.0/5 BST TON T4:96 0.001 500 0 NXB XIC T4:96/DN OTE B30:5/0 BND EOR
%   B30:0/0  EMO_INSTALLED  "CONFIG The EMO is installed" %
%   I:1.0/5  EMERGENCY_STOP  "EMO" %
%   T4:96  EMO_STARTUP_DELAY %
%   B30:5/0  EMO_ACTIVE  "STATUS The EMO has been depressed" %

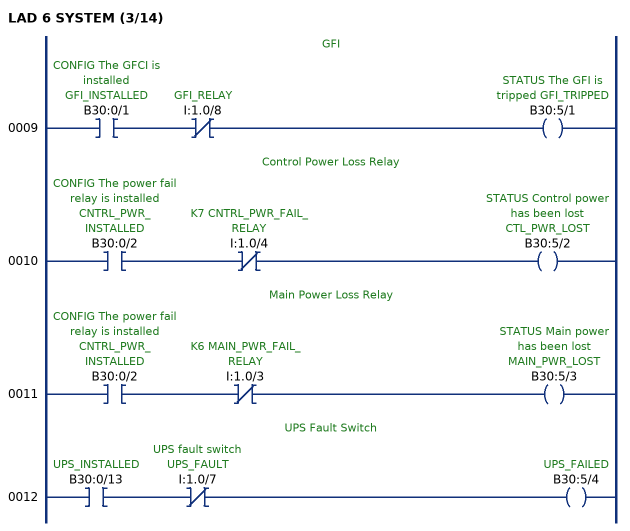
% Rung: 9 %
% GFI %
SOR XIC B30:0/1 XIO I:1.0/8 OTE B30:5/1 EOR
%   B30:0/1  GFI_INSTALLED  "CONFIG The GFCI is installed" %
%   I:1.0/8  GFI_RELAY %
%   B30:5/1  GFI_TRIPPED  "STATUS The GFI is tripped" %
% Rung: 10 %
% Control Power Loss Relay %
SOR XIC B30:0/2 XIO I:1.0/4 OTE B30:5/2 EOR
%   B30:0/2  CNTRL_PWR_INSTALLED  "CONFIG The power fail relay is installed" %
%   I:1.0/4  CNTRL_PWR_FAIL_RELAY  "K7" %
%   B30:5/2  CTL_PWR_LOST  "STATUS Control power has been lost" %
% Rung: 11 %
% Main Power Loss Relay %
SOR XIC B30:0/2 XIO I:1.0/3 OTE B30:5/3 EOR
%   B30:0/2  CNTRL_PWR_INSTALLED  "CONFIG The power fail relay is installed" %
%   I:1.0/3  MAIN_PWR_FAIL_RELAY  "K6" %
%   B30:5/3  MAIN_PWR_LOST  "STATUS Main power has been lost" %
% Rung: 12 %
% UPS Fault Switch %
SOR XIC B30:0/13 XIO I:1.0/7 OTE B30:5/4 EOR
%   B30:0/13  UPS_INSTALLED %
%   I:1.0/7  UPS_FAULT  "UPS fault switch" %
%   B30:5/4  UPS_FAILED %

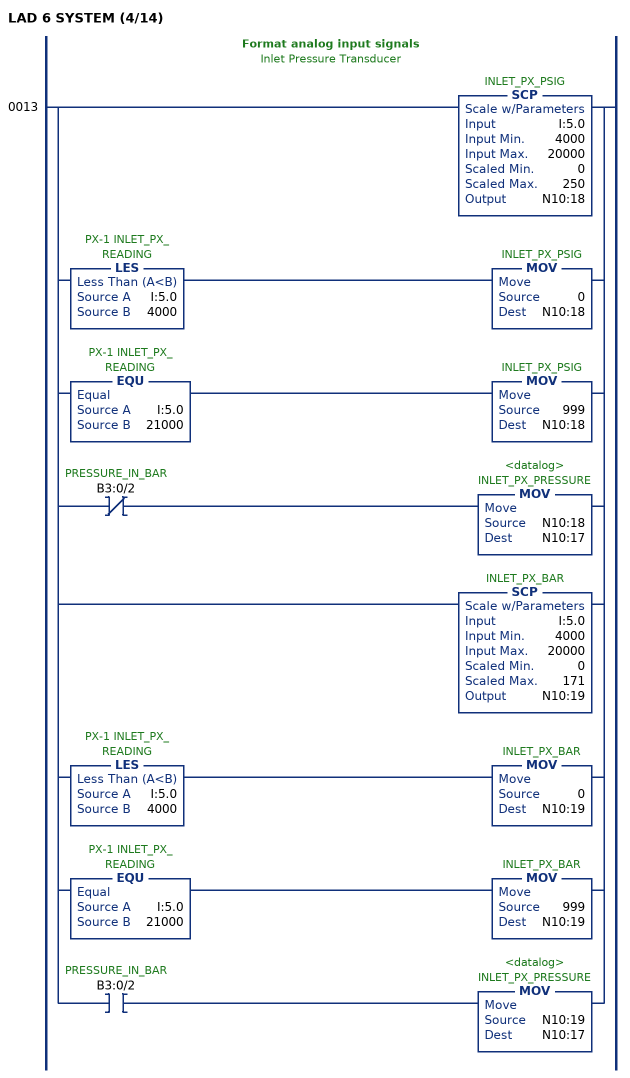
% Rung: 13 %
% TITLE: Format analog input signals %
% Inlet Pressure Transducer %
SOR BST SCP I:5.0 4000 20000 0 250 N10:18 NXB LES I:5.0 4000 MOV 0 N10:18 NXB EQU I:5.0 21000 MOV 999 N10:18 NXB XIO B3:0/2 MOV N10:18 N10:17 NXB SCP I:5.0 4000 20000 0 171 N10:19 NXB LES I:5.0 4000 MOV 0 N10:19 NXB EQU I:5.0 21000 MOV 999 N10:19 NXB XIC B3:0/2 MOV N10:19 N10:17 BND EOR
%   I:5.0  INLET_PX_READING  "PX-1" %
%   N10:18  INLET_PX_PSIG %
%   B3:0/2  PRESSURE_IN_BAR %
%   N10:17  INLET_PX_PRESSURE  "<datalog>" %
%   N10:19  INLET_PX_BAR %

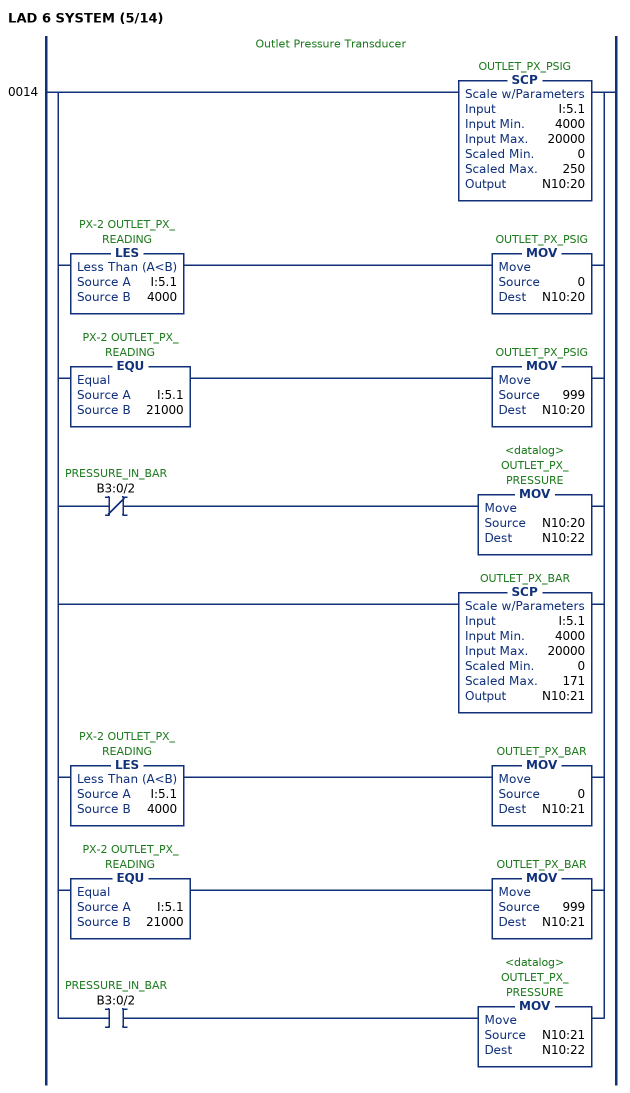
% Rung: 14 %
% Outlet Pressure Transducer %
SOR BST SCP I:5.1 4000 20000 0 250 N10:20 NXB LES I:5.1 4000 MOV 0 N10:20 NXB EQU I:5.1 21000 MOV 999 N10:20 NXB XIO B3:0/2 MOV N10:20 N10:22 NXB SCP I:5.1 4000 20000 0 171 N10:21 NXB LES I:5.1 4000 MOV 0 N10:21 NXB EQU I:5.1 21000 MOV 999 N10:21 NXB XIC B3:0/2 MOV N10:21 N10:22 BND EOR
%   I:5.1  OUTLET_PX_READING  "PX-2" %
%   N10:20  OUTLET_PX_PSIG %
%   B3:0/2  PRESSURE_IN_BAR %
%   N10:22  OUTLET_PX_PRESSURE  "<datalog>" %
%   N10:21  OUTLET_PX_BAR %

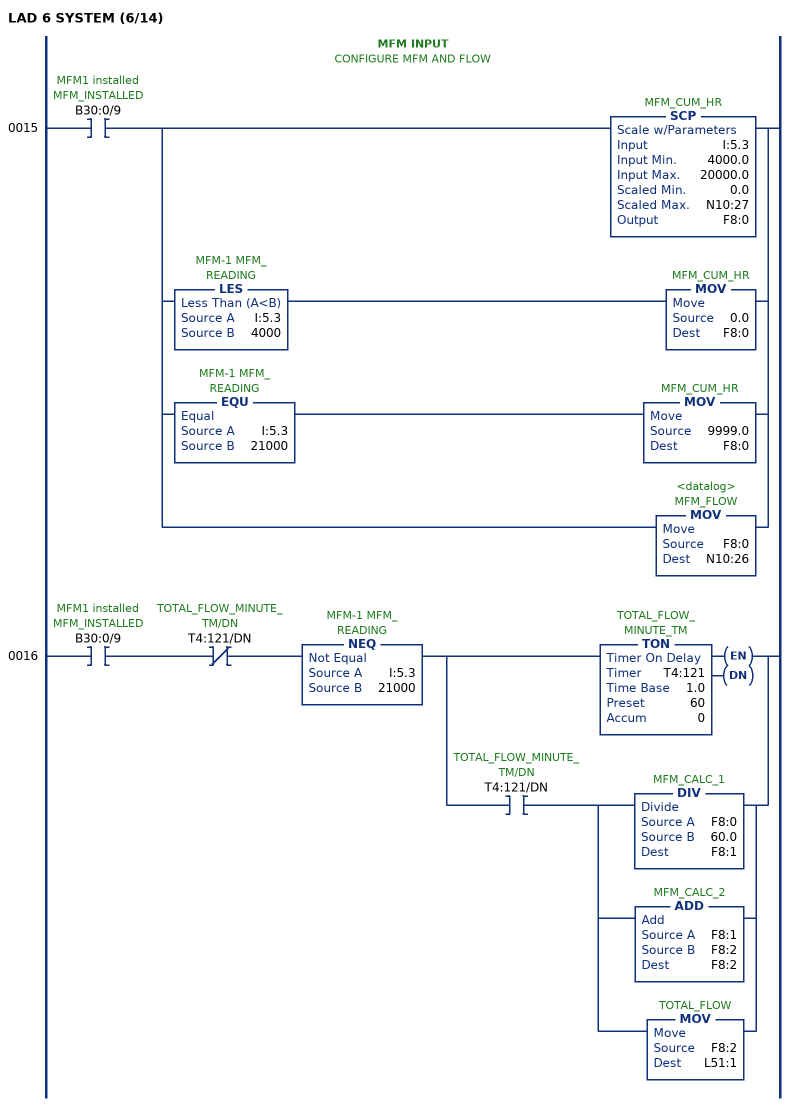
% Rung: 15 %
% TITLE: MFM INPUT %
% CONFIGURE MFM AND FLOW %
SOR XIC B30:0/9 BST SCP I:5.3 4000.0 20000.0 0.0 N10:27 F8:0 NXB LES I:5.3 4000 MOV 0.0 F8:0 NXB EQU I:5.3 21000 MOV 9999.0 F8:0 NXB MOV F8:0 N10:26 BND EOR
%   B30:0/9  MFM_INSTALLED  "MFM1 installed" %
%   I:5.3  MFM_READING  "MFM-1" %
%   N10:27  MFM_SCALING %
%   F8:0  MFM_CUM_HR %
%   N10:26  MFM_FLOW  "<datalog>" %
% Rung: 16 %
SOR XIC B30:0/9 XIO T4:121/DN NEQ I:5.3 21000 BST TON T4:121 1.0 60 0 NXB XIC T4:121/DN BST DIV F8:0 60.0 F8:1 NXB ADD F8:1 F8:2 F8:2 NXB MOV F8:2 L51:1 BND BND EOR
%   B30:0/9  MFM_INSTALLED  "MFM1 installed" %
%   T4:121  TOTAL_FLOW_MINUTE_TM %
%   I:5.3  MFM_READING  "MFM-1" %
%   F8:0  MFM_CUM_HR %
%   F8:1  MFM_CALC_1 %
%   F8:2  MFM_CALC_2 %
%   L51:1  TOTAL_FLOW %

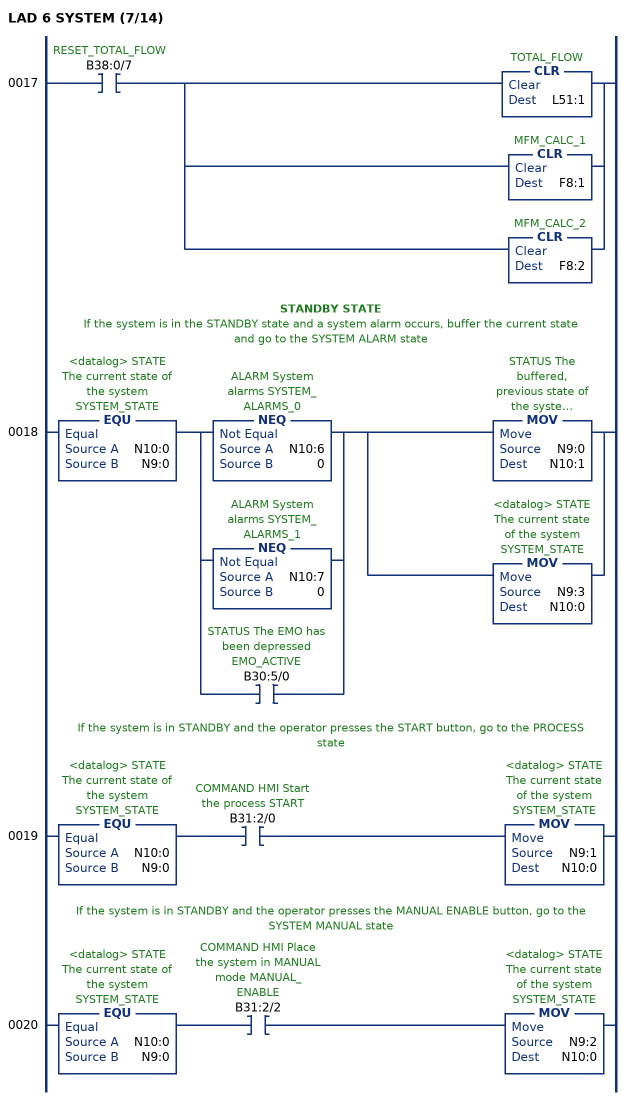
% Rung: 17 %
SOR XIC B38:0/7 BST CLR L51:1 NXB CLR F8:1 NXB CLR F8:2 BND EOR
%   B38:0/7  RESET_TOTAL_FLOW %
%   L51:1  TOTAL_FLOW %
%   F8:1  MFM_CALC_1 %
%   F8:2  MFM_CALC_2 %
% Rung: 18 %
% TITLE: STANDBY STATE %
% If the system is in the STANDBY state and a system alarm occurs, buffer the current state and go to the SYSTEM ALARM state %
SOR EQU N10:0 N9:0 BST NEQ N10:6 0 NXB NEQ N10:7 0 NXB XIC B30:5/0 BND BST MOV N9:0 N10:1 NXB MOV N9:3 N10:0 BND EOR
%   N10:0  SYSTEM_STATE  "<datalog> STATE The current state of the system" %
%   N9:0  SYSTEM_STANDBY  "STATE System Standby" %
%   N10:6  SYSTEM_ALARMS_0  "ALARM System alarms" %
%   N10:7  SYSTEM_ALARMS_1  "ALARM System alarms" %
%   B30:5/0  EMO_ACTIVE  "STATUS The EMO has been depressed" %
%   N10:1  SYSTEM_BUFFER  "STATUS The buffered, previous state of the system" %
%   N9:3  SYSTEM_ALARM  "STATE System Alarm" %
% Rung: 19 %
% If the system is in STANDBY and the operator presses the START button, go to the PROCESS state %
SOR EQU N10:0 N9:0 XIC B31:2/0 MOV N9:1 N10:0 EOR
%   N10:0  SYSTEM_STATE  "<datalog> STATE The current state of the system" %
%   N9:0  SYSTEM_STANDBY  "STATE System Standby" %
%   B31:2/0  START  "COMMAND HMI Start the process" %
%   N9:1  SYSTEM_PROCESS  "STATE System Process" %
% Rung: 20 %
% If the system is in STANDBY and the operator presses the MANUAL ENABLE button, go to the SYSTEM MANUAL state %
SOR EQU N10:0 N9:0 XIC B31:2/2 MOV N9:2 N10:0 EOR
%   N10:0  SYSTEM_STATE  "<datalog> STATE The current state of the system" %
%   N9:0  SYSTEM_STANDBY  "STATE System Standby" %
%   B31:2/2  MANUAL_ENABLE  "COMMAND HMI Place the system in MANUAL mode" %
%   N9:2  SYSTEM_MANUAL  "STATE System Manual" %

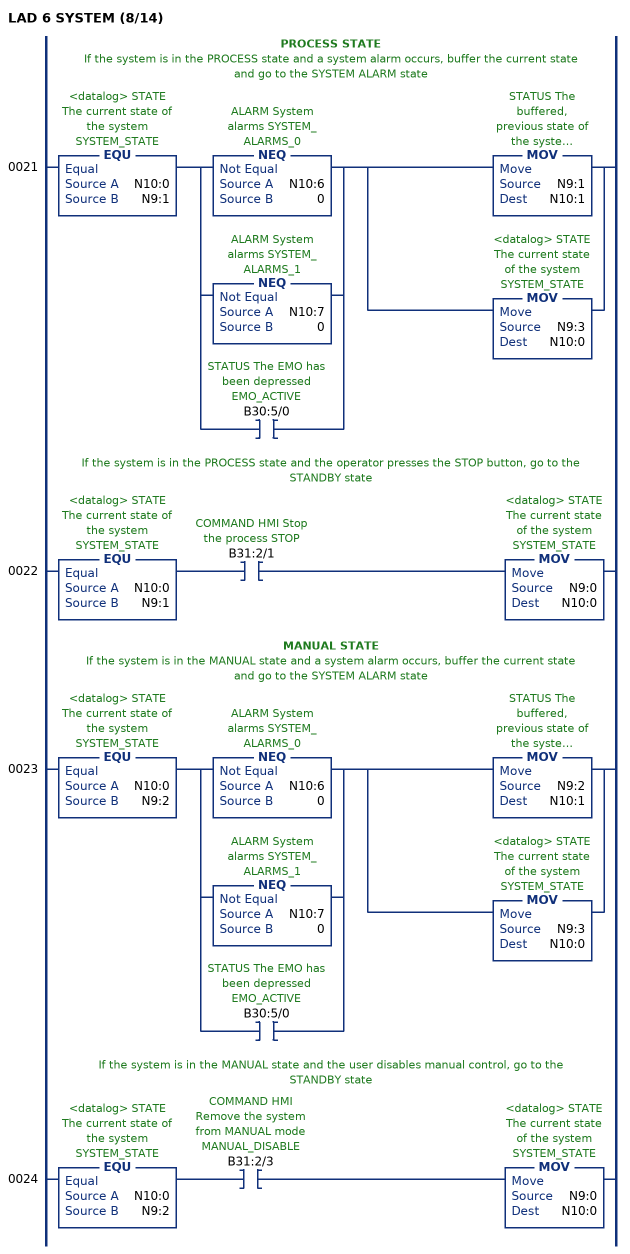
% Rung: 21 %
% TITLE: PROCESS STATE %
% If the system is in the PROCESS state and a system alarm occurs, buffer the current state and go to the SYSTEM ALARM state %
SOR EQU N10:0 N9:1 BST NEQ N10:6 0 NXB NEQ N10:7 0 NXB XIC B30:5/0 BND BST MOV N9:1 N10:1 NXB MOV N9:3 N10:0 BND EOR
%   N10:0  SYSTEM_STATE  "<datalog> STATE The current state of the system" %
%   N9:1  SYSTEM_PROCESS  "STATE System Process" %
%   N10:6  SYSTEM_ALARMS_0  "ALARM System alarms" %
%   N10:7  SYSTEM_ALARMS_1  "ALARM System alarms" %
%   B30:5/0  EMO_ACTIVE  "STATUS The EMO has been depressed" %
%   N10:1  SYSTEM_BUFFER  "STATUS The buffered, previous state of the system" %
%   N9:3  SYSTEM_ALARM  "STATE System Alarm" %
% Rung: 22 %
% If the system is in the PROCESS state and the operator presses the STOP button, go to the STANDBY state %
SOR EQU N10:0 N9:1 XIC B31:2/1 MOV N9:0 N10:0 EOR
%   N10:0  SYSTEM_STATE  "<datalog> STATE The current state of the system" %
%   N9:1  SYSTEM_PROCESS  "STATE System Process" %
%   B31:2/1  STOP  "COMMAND HMI Stop the process" %
%   N9:0  SYSTEM_STANDBY  "STATE System Standby" %
% Rung: 23 %
% TITLE: MANUAL STATE %
% If the system is in the MANUAL state and a system alarm occurs, buffer the current state and go to the SYSTEM ALARM state %
SOR EQU N10:0 N9:2 BST NEQ N10:6 0 NXB NEQ N10:7 0 NXB XIC B30:5/0 BND BST MOV N9:2 N10:1 NXB MOV N9:3 N10:0 BND EOR
%   N10:0  SYSTEM_STATE  "<datalog> STATE The current state of the system" %
%   N9:2  SYSTEM_MANUAL  "STATE System Manual" %
%   N10:6  SYSTEM_ALARMS_0  "ALARM System alarms" %
%   N10:7  SYSTEM_ALARMS_1  "ALARM System alarms" %
%   B30:5/0  EMO_ACTIVE  "STATUS The EMO has been depressed" %
%   N10:1  SYSTEM_BUFFER  "STATUS The buffered, previous state of the system" %
%   N9:3  SYSTEM_ALARM  "STATE System Alarm" %
% Rung: 24 %
% If the system is in the MANUAL state and the user disables manual control, go to the STANDBY state %
SOR EQU N10:0 N9:2 XIC B31:2/3 MOV N9:0 N10:0 EOR
%   N10:0  SYSTEM_STATE  "<datalog> STATE The current state of the system" %
%   N9:2  SYSTEM_MANUAL  "STATE System Manual" %
%   B31:2/3  MANUAL_DISABLE  "COMMAND HMI Remove the system from MANUAL mode" %
%   N9:0  SYSTEM_STANDBY  "STATE System Standby" %

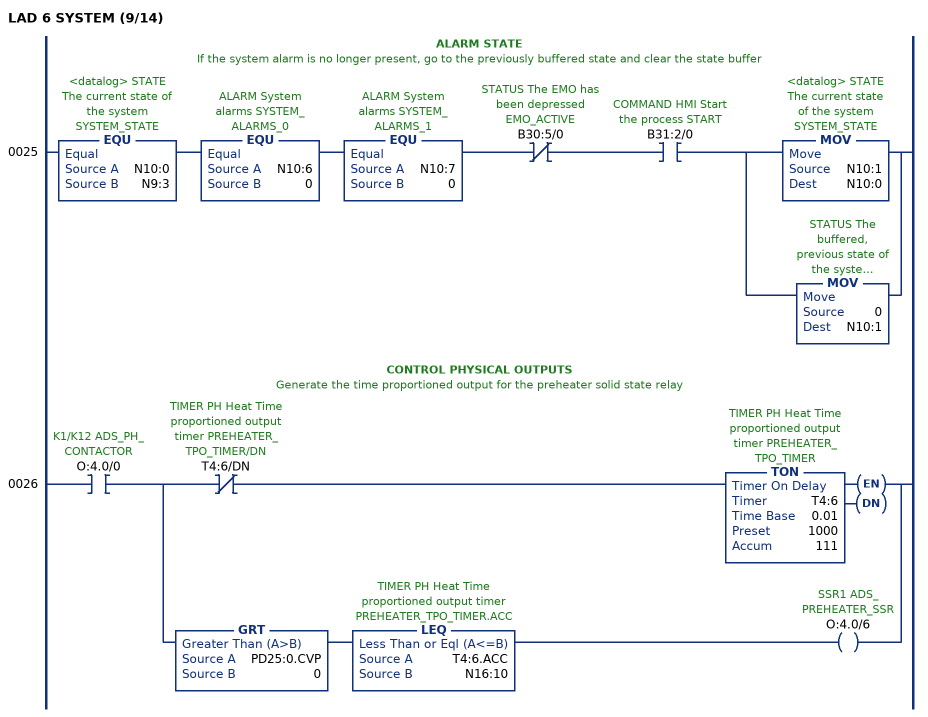
% Rung: 25 %
% TITLE: ALARM STATE %
% If the system alarm is no longer present, go to the previously buffered state and clear the state buffer %
SOR EQU N10:0 N9:3 EQU N10:6 0 EQU N10:7 0 XIO B30:5/0 XIC B31:2/0 BST MOV N10:1 N10:0 NXB MOV 0 N10:1 BND EOR
%   N10:0  SYSTEM_STATE  "<datalog> STATE The current state of the system" %
%   N9:3  SYSTEM_ALARM  "STATE System Alarm" %
%   N10:6  SYSTEM_ALARMS_0  "ALARM System alarms" %
%   N10:7  SYSTEM_ALARMS_1  "ALARM System alarms" %
%   B30:5/0  EMO_ACTIVE  "STATUS The EMO has been depressed" %
%   B31:2/0  START  "COMMAND HMI Start the process" %
%   N10:1  SYSTEM_BUFFER  "STATUS The buffered, previous state of the system" %
% Rung: 26 %
% TITLE: CONTROL PHYSICAL OUTPUTS %
% Generate the time proportioned output for the preheater solid state relay %
SOR XIC O:4.0/0 BST XIO T4:6/DN TON T4:6 0.01 1000 111 NXB GRT PD25:0.CVP 0 LEQ T4:6.ACC N16:10 OTE O:4.0/6 BND EOR
%   O:4.0/0  ADS_PH_CONTACTOR  "K1/K12" %
%   T4:6  PREHEATER_TPO_TIMER  "TIMER PH Heat Time proportioned output timer" %
%   N16:10  ADS_PH_OUTPUT  "<datalog> CONTROL ADS Preheater output (percent)" %
%   O:4.0/6  ADS_PREHEATER_SSR  "SSR1" %

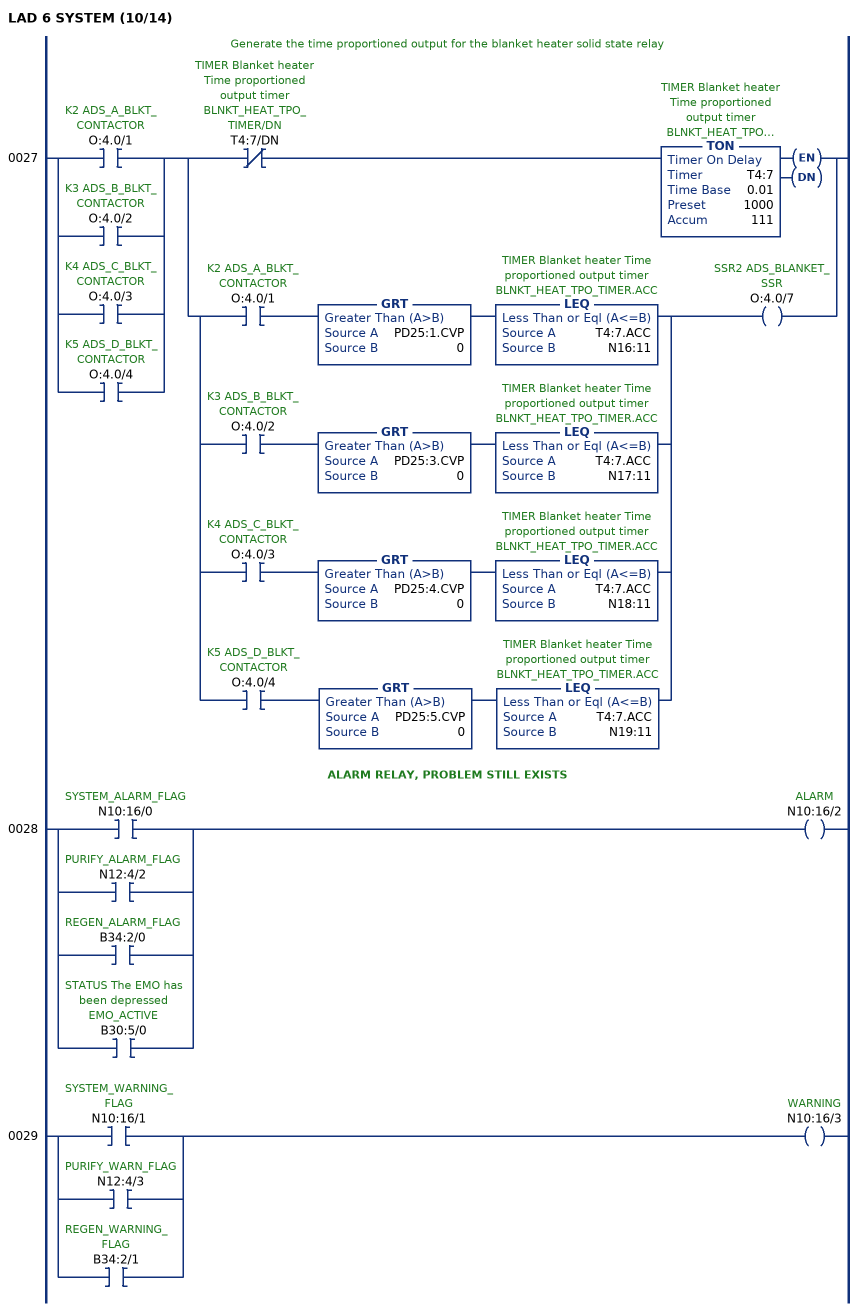
% Rung: 27 %
% Generate the time proportioned output for the blanket heater solid state relay %
SOR BST XIC O:4.0/1 NXB XIC O:4.0/2 NXB XIC O:4.0/3 NXB XIC O:4.0/4 BND BST XIO T4:7/DN TON T4:7 0.01 1000 111 NXB BST XIC O:4.0/1 GRT PD25:1.CVP 0 LEQ T4:7.ACC N16:11 NXB XIC O:4.0/2 GRT PD25:3.CVP 0 LEQ T4:7.ACC N17:11 NXB XIC O:4.0/3 GRT PD25:4.CVP 0 LEQ T4:7.ACC N18:11 NXB XIC O:4.0/4 GRT PD25:5.CVP 0 LEQ T4:7.ACC N19:11 BND OTE O:4.0/7 BND EOR
%   O:4.0/1  ADS_A_BLKT_CONTACTOR  "K2" %
%   O:4.0/2  ADS_B_BLKT_CONTACTOR  "K3" %
%   O:4.0/3  ADS_C_BLKT_CONTACTOR  "K4" %
%   O:4.0/4  ADS_D_BLKT_CONTACTOR  "K5" %
%   T4:7  BLNKT_HEAT_TPO_TIMER  "TIMER Blanket heater Time proportioned output timer" %
%   N16:11  ADS_A_BLNKT_OUTPUT  "<datalog> CONTROL ADS A Blanket output (percent)" %
%   N17:11  ADS_B_BLNKT_OUTPUT  "<datalog> CONTROL ADS A Blanket output" %
%   N18:11  ADS_C_BLNKT_OUTPUT  "<datalog>" %
%   N19:11  ADS_D_BLNKT_OUTPUT  "<datalog>" %
%   O:4.0/7  ADS_BLANKET_SSR  "SSR2" %
% Rung: 28 %
% TITLE: ALARM RELAY, PROBLEM STILL EXISTS %
SOR BST XIC N10:16/0 NXB XIC N12:4/2 NXB XIC B34:2/0 NXB XIC B30:5/0 BND OTE N10:16/2 EOR
%   N10:16/0  SYSTEM_ALARM_FLAG %
%   N12:4/2  PURIFY_ALARM_FLAG %
%   B34:2/0  REGEN_ALARM_FLAG %
%   B30:5/0  EMO_ACTIVE  "STATUS The EMO has been depressed" %
%   N10:16/2  ALARM %
% Rung: 29 %
SOR BST XIC N10:16/1 NXB XIC N12:4/3 NXB XIC B34:2/1 BND OTE N10:16/3 EOR
%   N10:16/1  SYSTEM_WARNING_FLAG %
%   N12:4/3  PURIFY_WARN_FLAG %
%   B34:2/1  REGEN_WARNING_FLAG %
%   N10:16/3  WARNING %

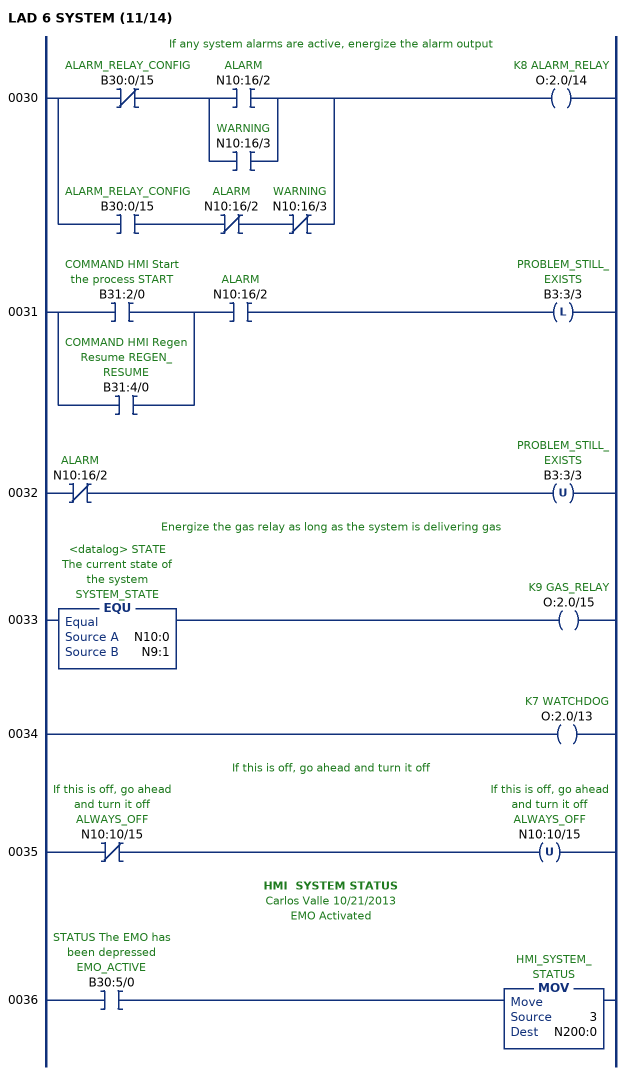
% Rung: 30 %
% If any system alarms are active, energize the alarm output %
SOR BST XIO B30:0/15 BST XIC N10:16/2 NXB XIC N10:16/3 BND NXB XIC B30:0/15 XIO N10:16/2 XIO N10:16/3 BND OTE O:2.0/14 EOR
%   B30:0/15  ALARM_RELAY_CONFIG %
%   N10:16/2  ALARM %
%   N10:16/3  WARNING %
%   O:2.0/14  ALARM_RELAY  "K8" %
% Rung: 31 %
SOR BST XIC B31:2/0 NXB XIC B31:4/0 BND XIC N10:16/2 OTL B3:3/3 EOR
%   B31:2/0  START  "COMMAND HMI Start the process" %
%   B31:4/0  REGEN_RESUME  "COMMAND HMI Regen Resume" %
%   N10:16/2  ALARM %
%   B3:3/3  PROBLEM_STILL_EXISTS %
% Rung: 32 %
SOR XIO N10:16/2 OTU B3:3/3 EOR
%   N10:16/2  ALARM %
%   B3:3/3  PROBLEM_STILL_EXISTS %
% Rung: 33 %
% Energize the gas relay as long as the system is delivering gas %
SOR EQU N10:0 N9:1 OTE O:2.0/15 EOR
%   N10:0  SYSTEM_STATE  "<datalog> STATE The current state of the system" %
%   N9:1  SYSTEM_PROCESS  "STATE System Process" %
%   O:2.0/15  GAS_RELAY  "K9" %
% Rung: 34 %
SOR OTE O:2.0/13 EOR
%   O:2.0/13  WATCHDOG  "K7" %
% Rung: 35 %
% If this is off, go ahead and turn it off %
SOR XIO N10:10/15 OTU N10:10/15 EOR
%   N10:10/15  ALWAYS_OFF  "If this is off, go ahead and turn it off" %
% Rung: 36 %
% TITLE: HMI  SYSTEM STATUS %
% Carlos Valle 10/21/2013
% EMO Activated %
SOR XIC B30:5/0 MOV 3 N200:0 EOR
%   B30:5/0  EMO_ACTIVE  "STATUS The EMO has been depressed" %
%   N200:0  HMI_SYSTEM_STATUS %

